{attribute 'qualified_only'}
VAR_GLOBAL

END_VAR

(* stored: Version 1.1.0.1, ProductVersion 3.1.4024.12
   GVL Globals: Id {0134dc14-cb11-4017-ba71-6922c72c5567} *)
